FUNCTION_BLOCK Junction
VAR_IN_OUT
	conveyor1 : ConveyorLSC;
	conveyor2 : ConveyorLSC;
	conveyor3 : ConveyorLSC;
	conveyor4 : ConveyorLSC;
	conveyor5 : ConveyorLSC;
	conveyor6 : ConveyorLSC;
END_VAR
VAR
	nextBuffer : POINTER TO IndexedBuffer;
	prevBuffer : POINTER TO IndexedBuffer;
	
	conveyors : ARRAY[1..CONSTS.numConveyorLines] OF POINTER TO ConveyorSC;
	iBundles : ARRAY[1..CONSTS.numConveyorLines] OF INT := [6(-1)];
	
	step : SectionTask;
END_VAR

CASE step OF
	SectionTask.IDLE:
		
		
	SectionTask.ALIGN:
		
		
	SectionTask.ACTIVE:
		(*
		1	send all bundles that do no need area transfer over the junction 
			-iterate through array of iterators
				*if bundle does not need transfer then request the conveyor FWD
				*if bundle needs transfer, then hold the conveyor
			
		2	 
		*)
	
	
END_CASE

END_FUNCTION_BLOCK

(* stored: Version 1.1.0.1, ProductVersion 3.1.4024.11
   POU Junction: Id {7e1335d0-8c31-4598-8596-1c04f880fb59}, SpecialFunc None *)
